FUNCTION_BLOCK EL5002
VAR
	_io : EL5002_Data;
	{attribute addProperty Name "WcState"}
	_wcState : WcStateInputToggle;
	{attribute addProperty Name "Info data"}
	_infoData : InfoDataAdsDC;
END_VAR

PROPERTY IO : REFERENCE TO EL5002_Data
GET
IO REF= _io;
END_GET
END_PROPERTY

PROPERTY WcState : REFERENCE TO WcStateInputToggle
GET
WcState REF= _wcState;
END_GET
END_PROPERTY

END_FUNCTION_BLOCK

(* stored: Version 1.1.0.1, ProductVersion 3.1.4024.9
   POU EL5002: Id {f1ef9e2a-5816-04a5-2a4e-220b8bfc92f1}, SpecialFunc None
   Property IO: Id {eb63913b-edae-03f3-08f9-bdeb36f4103a}
   Get Get: Id {25bc21e7-482b-0d85-1722-39a01ea394ac}
   Property WcState: Id {f903842d-d18e-0e4f-35eb-75f05b3eefd1}
   Get Get: Id {65c70a6b-f893-09c7-030a-6bf8df1c5a11} *)
